// TIA Portal V16 export
// export: Created 2024-12-03T15:41:45.1170652Z, ExportSetting WithReadOnly, DisplayName Totally Integrated Automation Portal, DisplayVersion V16 Update 6, DisplayName TIA Portal Version Control Interface, DisplayVersion V16 Update 2, DisplayName TIA Portal Openness, DisplayVersion V16 Update 6, DisplayName TIA Portal Teamcenter Gateway, DisplayVersion V16, DisplayName SINAMICS Startdrive Advanced, DisplayVersion V16 Update 5, DisplayName SINAMICS Startdrive G130, G150, S120, S150, SINAMICS MV, S210, DisplayVersion V16 Update 5, DisplayName SINAMICS Startdrive G110M, G120, G120C, G120D, G120P, G115D, DisplayVersion V16 Update 5, DisplayName STEP 7 Professional, DisplayVersion V16 Update 6, DisplayName STEP 7 Safety, DisplayVersion V16, DisplayName WinCC Advanced / Unified PC, DisplayVersion V16 Update 6
TYPE "Scale_UDT"
// stored: CreationDate 2021-07-13T07:41:36.2278727Z, InterfaceModifiedDate 2023-08-01T07:36:31.0856308Z, IsConsistent true, LibraryConformanceStatus The object is library-conformant., ModifiedDate 2023-08-01T07:36:31.0856308Z
   STRUCT
      Cmd : Struct
         Reset : Bool;
         ResetDiagnostics : Bool;
         Manual : "Scale_CMD_UDT";
         Auto : "Scale_CMD_UDT";
      END_STRUCT;
      settings : Struct
         offset : Real;
         stabWeight : Real;
         stabilizationTime : Time;
      END_STRUCT;
      status : Struct
         ManualModeActive : Bool;
         ReadyForNewCommand : Bool;   // Ready”, thus status indicates a new command can be done. This includes “Zero”, “Tare”, “ResetTare” and “Command” inputs parameters. If you use other add-on instructions, the “Ready” status can also change when other blocs send commands to the scale. It is recommended to test “Ready” status before sending a command
         ExecutingCommand : Bool;
         GrossWeight : Real;
         NetWeight : Real;
      END_STRUCT;
      diagnostics : Struct
         stableMeasurements : DInt;
         unstableMeasurements : DInt;
         totalMeasurements : DInt;
      END_STRUCT;
      ReadResult : Struct
         NewResult : Bool;
         NewResult_Flag : Bool;
         Stable : Bool;
         netWeightGrams : DInt;
         netWeightGrams_Flag : DInt;
      END_STRUCT;
      alarms : Struct
         Error : "HmiAlarm";
         notConnected : "HmiAlarm";
         Status { S7_SetPoint := 'True'} : Word;
      END_STRUCT;
      "Name" : String[40];
      zone : Int;
   END_STRUCT;
END_TYPE
